TYPE ST_M001_IO :
STRUCT
	stIn 	AT%I* : ST_M001_IO_IN;
	stOut 	AT%Q* : ST_M001_IO_OUT;
END_STRUCT
END_TYPE

(* stored: Version 1.1.0.1
   DUT ST_M001_IO: Id {7734a3f4-177d-4cfe-a519-7734878c0bef} *)
